// TIA Portal project "PIONEER" (V19)

(* hardware
DEVICE "S7-1500/ET200MP station_1"  S7-1500 station
   slot 0: "Rail_0"  Rack  6ES7 590-1***0-0AA0
   slot 1: "PLC_1"  CPU 1516F-3 PN/DP  6ES7 516-3FN01-0AB0  V2.6
      slot 3: "CPU display_1"  6ES7591-1BA00-0AA0
      slot 32768: "PROFINET interface_1"  X1
         slot 32769: "Port_1"  X1 P1
         slot 32770: "Port_2"  X1 P2
      slot 33024: "PROFINET interface_2"  X2
         slot 33025: "Port_1"  X2 P1
      slot 33280: "DP interface_1"  X3
   slot 2: "DI 32x24VDC HF_1"  DI 32x24VDC HF  6ES7 521-1BL00-0AB0  V2.2
   slot 3: "DQ 32x24VDC/0.5A ST_1"  DQ 32x24VDC/0.5A ST  6ES7 522-1BL00-0AB0  V2.0
   slot 4: "AI 8xU/I/RTD/TC ST_1"  AI 8xU/I/RTD/TC ST  6ES7 531-7KF00-0AB0  V2.2
   slot 5: "AQ 4xU/I ST_1"  AQ 4xU/I ST  6ES7 532-5HD00-0AB0  V2.2
DEVICE "S7-1200 station_1"  S7-1200 Station
   slot 0: "Rack_0"  S7-1200 Rack  Rack  V1.0
   slot 1: "PLC_2"  CPU 1214C DC/DC/DC  6ES7 214-1AG40-0XB0  V4.2
   slot 2: "DI 8/DQ 8x24VDC_1"  6ES7 223-1BH32-0XB0  V2.0
   slot 3: "AQ 1x12BIT_1"  AQ1 signal board  6ES7 232-4HA30-0XB0  V1.0
*)

// ===== PLC "PLC_1"  CPU 1516F-3 PN/DP =====

VAR_GLOBAL   // PLC tag table "Default tag table"
   "gestures" AT %MB0 : Byte;
   "LightSensorCube" AT %I0.0 : Bool;
   "LightSensorCylinder" AT %I0.1 : Bool;
   "LightSensorWorkpiece" AT %I0.2 : Bool;
   "LimitSwitchCylinderNotExtended" AT %I0.3 : Bool;
   "LimitSwitchCylinderRetracted" AT %I0.4 : Bool;
   "WorkpieceCylinder" AT %Q0.0 : Bool;
   "WorkpieceCube" AT %Q0.1 : Bool;
   "CylinderHeadRetract" AT %Q0.2 : Bool;
   "CylinderHeadExtend" AT %Q0.3 : Bool;
   "ConveyorLong" AT %Q0.4 : Bool;
   "ConveyorShort" AT %Q0.5 : Bool;
END_VAR

DATA_BLOCK "Main_Safety_RTG1_DB"   // DB1, F_DB
{ S7_Optimized_Access := 'TRUE' }
NAME : FUSI
VERSION : 0.1
// stored: InstanceOfName Main_Safety_RTG1
"Main_Safety_RTG1"
BEGIN
END_DATA_BLOCK

DATA_BLOCK "Gesture_Pioneer_DB"   // DB2
{ S7_Optimized_Access := 'TRUE' }
VERSION : 0.1
// stored: InstanceOfName Gesture_Pioneer
"Gesture_Pioneer"
BEGIN
END_DATA_BLOCK

FUNCTION_BLOCK "Main_Safety_RTG1"   // FB1, F_FBD
{ S7_Optimized_Access := 'TRUE' }
BEGIN
END_FUNCTION_BLOCK

FUNCTION_BLOCK "Gesture_Pioneer"   // FB2, SCL
{ S7_Optimized_Access := 'TRUE' }
VERSION : 0.1
   VAR
      "STEP" : Int;
   END_VAR
BEGIN
   CASE #STEP OF
       0: 
           IF "gestures".%X1 THEN
               "ConveyorShort" := 1;
           ELSIF "gestures".%X0 THEN
               "ConveyorLong" := 1;
           ELSIF "gestures".%X2 THEN
               "ConveyorShort" := 0;
           ELSIF "gestures".%X3 THEN
               "ConveyorLong" := 0;
           ELSIF "gestures".%X4 THEN
               "WorkpieceCube" := 1;
               "WorkpieceCylinder" := 1;
           END_IF;
   END_CASE;
END_FUNCTION_BLOCK

ORGANIZATION_BLOCK "Main"   // OB1, LAD, ProgramCycle
TITLE = "Main Program Sweep (Cycle)"
{ S7_Optimized_Access := 'TRUE' }
VERSION : 0.1
   VAR_INPUT
      Initial_Call : Bool;   // Initial call of this OB
      Remanence : Bool;   // =True, if remanent data are available
   END_VAR
BEGIN

REGION Network 1
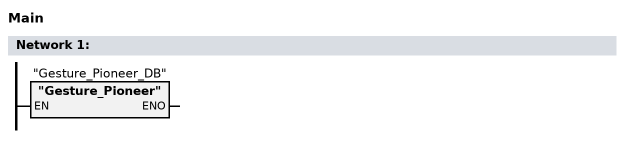
   RUNG wire#powerrail
      "Gesture_Pioneer_DB"()
   END_RUNG
   // the same network as SCL:
   "Gesture_Pioneer_DB"();   // "Gesture_Pioneer"
END_REGION
END_ORGANIZATION_BLOCK

// ===== PLC "PLC_2"  CPU 1214C DC/DC/DC =====

VAR_GLOBAL   // PLC tag table "Default tag table"
   "whatever" AT %MB0 : Byte;
   "Foward" AT %Q0.0 : Bool;
   "Backward" AT %Q0.1 : Bool;
END_VAR

DATA_BLOCK "Gesture_DB"   // DB1
{ S7_Optimized_Access := 'TRUE' }
VERSION : 0.1
// stored: InstanceOfName Gesture
"Gesture"
BEGIN
END_DATA_BLOCK

FUNCTION_BLOCK "Gesture"   // FB1, SCL
{ S7_Optimized_Access := 'TRUE' }
VERSION : 0.1
   VAR
      "STEP" : Bool;
   END_VAR
BEGIN
   IF "whatever".%X1 THEN
       "Foward" := true;
       "Backward" := FALSE;
   END_IF;
   IF "whatever".%X0 THEN
       "Foward" := FALSE;
       "Backward" := TRUE;
   END_IF;
END_FUNCTION_BLOCK

ORGANIZATION_BLOCK "Main"   // OB1, LAD, ProgramCycle
TITLE = "Main Program Sweep (Cycle)"
{ S7_Optimized_Access := 'TRUE' }
VERSION : 0.1
   VAR_INPUT
      Initial_Call : Bool;   // Initial call of this OB
      Remanence : Bool;   // =True, if remanent data are available
   END_VAR
BEGIN

REGION Network 1
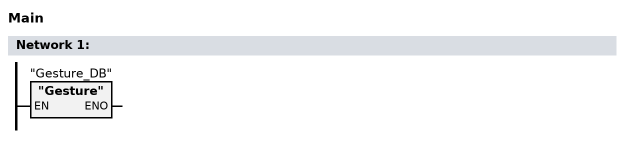
   RUNG wire#powerrail
      "Gesture_DB"()
   END_RUNG
   // the same network as SCL:
   "Gesture_DB"();   // "Gesture"
END_REGION
END_ORGANIZATION_BLOCK